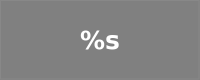
VISUALIZATION MenuItem  // 200x80
VAR_INPUT
	i_nFrameNumber : DINT;
	i_sText : STRING;
	i_itfVisuMenu : ITF_Visu_Menu;
END_VAR
VAR
	dwElemColor			: DWORD := 16#FF808080;
	dwDarkGray			: DWORD := 16#FF808080; // Decimal R128 G128 B128
	dwLightGray			: DWORD := 16#FFDCDCDC; // Decimal R220 G220 B220
	dwGray				: DWORD := 16#FFC8C8C8; // Decimal R200 R200 R200
	dwGrayHowover		: DWORD := 16#FF969696; // Decimal R150 G150 B150
END_VAR
    Rectangle (0,0 200x80), "%s", text variable: i_sText, colour toggle: i_itfVisuMenu.Page = FrameNumber
    Rectangle (0,0 200x80), colour toggle: i_itfVisuMenu.p_nPage = i_nFrameNumber
        OnMouseClick: execute { i_itfVisuMenu.m_SetPage(FrameNumber); dwElemColor := dwDarkGray; }
END_VISUALIZATION

(* stored: Version 1.1.0.1, ProductVersion 3.1.4026.13
   Visu MenuItem: Id {5159f1db-c9e5-477e-8bc2-cbc316391e8c} *)
